(* CoDeSys 2.3 export: TYPE_OUTPUTS.EXP *)

(* Data type *)
TYPE TYPE_OUTPUTS :
	STRUCT
		LEDAusgefahren: BOOL;
		LEDEingefahren: BOOL;
		LEDMontagePos: BOOL;
		RelaisMotorLeistung: BOOL;
		SchuetzGrundlast: BOOL;
	END_STRUCT
END_TYPE
